FUNCTION_BLOCK ABSTRACT fbSimpleRemoteExec
VAR
	_start : UINT;
	_done : UINT;
END_VAR

METHOD ABSTRACT Execute : BOOL
VAR_INPUT
	param : ANY;
END_VAR
END_METHOD

METHOD PUBLIC FINAL Invoke : BOOL
IF(THIS^._start > THIS^._done) THEN
	Execute();
END_IF
END_METHOD

END_FUNCTION_BLOCK

(* stored: Version 1.1.0.1, ProductVersion 3.1.4024.3
   POU fbSimpleRemoteExec: Id {43ea00d1-283e-4198-bb16-45f6cfaf4aeb}, SpecialFunc None
   Method Execute: Id {67b64cdb-f03d-4afd-bbb0-60eddd5e536d}
   Method Invoke: Id {716080f8-813f-4a50-8132-090c6e25e131} *)
